FUNCTION_BLOCK FB_ControlledValve EXTENDS FB_ActorContinous
VAR_INPUT
END_VAR
VAR_OUTPUT
END_VAR
VAR	
	bFeedbackSignal : BOOL := FALSE; //True if a feedback signal is provided	

	//I/O Links
	fActualPosition 	AT %I* : REAL; //Actual valve position
	
END_VAR

//Outputs
//Output (On/Off) := bSetStatusOn;

MAIN();

METHOD PROTECTED   SetState : BOOL
VAR_INPUT
END_VAR
//Set control state
IF bFeedbackSignal = TRUE THEN //Use feedback signal if possible
	IF fActualPosition > 0 THEN //Float signal must be greater than zero	
		controlState.bStatusOn := TRUE; 
	END_IF;
END_IF;

//set setpoint state
setPointState.fOperatingPoint := fActualPosition;

//Outputs
//Output (On/Off) := fSetPoint;
END_METHOD

END_FUNCTION_BLOCK

(* stored: Version 1.1.0.1, ProductVersion 3.1.4024.9
   POU FB_ControlledValve: Id {60dbc338-d028-4fcc-a2a7-9fe749ce4d3c}, SpecialFunc None
   Method SetState: Id {be832a62-70d4-4ec0-8ee4-578237454401} *)
